// LS Electric XG5000 project: Sincronismo com leitura da frequência real e correção automática pelo CLP
// PLC Main

PROGRAM NewProgram (task: Scan Program)

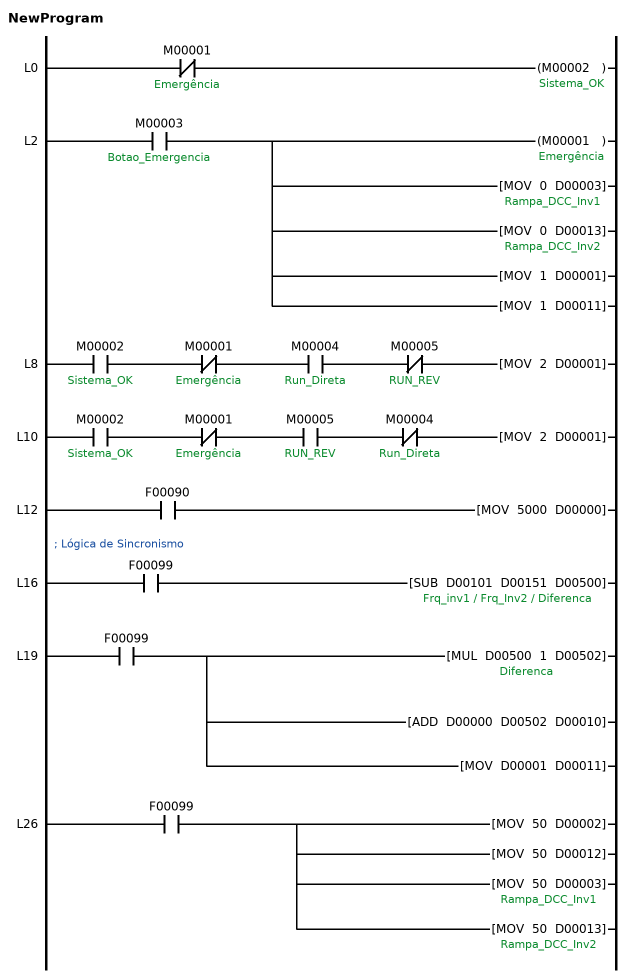
; L0
LOAD NOT  M00001	// Emergência
OUT       M00002	// Sistema_OK
; L2
LOAD      M00003	// Botao_Emergencia
OUT       M00001	// Emergência
MOV       0 D00003	// Rampa_DCC_Inv1
MOV       0 D00013	// Rampa_DCC_Inv2
MOV       1 D00001
MOV       1 D00011
; L8
LOAD      M00002	// Sistema_OK
AND NOT   M00001	// Emergência
AND       M00004	// Run_Direta
AND NOT   M00005	// RUN_REV
MOV       2 D00001
; L10
LOAD      M00002	// Sistema_OK
AND NOT   M00001	// Emergência
AND       M00005	// RUN_REV
AND NOT   M00004	// Run_Direta
MOV       2 D00001
; L12
LOAD      F00090
MOV       5000 D00000
// Lógica de Sincronismo
; L16
LOAD      F00099
SUB       D00101 D00151 D00500	// Frq_inv1 / Frq_Inv2 / Diferenca
; L19
LOAD      F00099
MUL       D00500 1 D00502	// Diferenca
ADD       D00000 D00502 D00010
MOV       D00001 D00011
; L26
LOAD      F00099
MOV       50 D00002
MOV       50 D00012
MOV       50 D00003	// Rampa_DCC_Inv1
MOV       50 D00013	// Rampa_DCC_Inv2